VAR
	iCount		: INT;
	apply_on	: BOOL;
END_VAR
    Rectangle (127,314 451x90)
    Rectangle (578,0 127x404)
    Rectangle (127,83 451x231)
    Rectangle (127,0 451x83)
    Rectangle (0,0 127x404)
    Label (134,42 113x38), "Производитель- ность, 0-100 %"
    Label (362,42 103x34), "Скорость ТЯУ, 0-100 %"
    RoundedRectangle (472,45 80x32), "%.1f", text variable: REG_ED.Speed
        OnMouseClick: write the text variable via VisuDialogs.Numpad, min QM_MIN, max QM_MAX, title "Производительность, %"
        OnMouseClick: execute { apply_on:=TRUE; }
    RoundedRectangle (31,14 80x32), "%.1f", text variable: REG_ED.TEMPS[0]
        OnMouseClick: write the text variable via VisuDialogs.Numpad, min T_MINS_ZAD[0], max T_MAXS_ZAD[0], title "ТЕМПЕРАТУРА 1 ЗОНЫ"
        OnMouseClick: execute { apply_on:=TRUE; }
    Label (4,17 40x20), "T1"
    RoundedRectangle (31,57 80x32), "%.1f", text variable: REG_ED.TEMPS[1]
        OnMouseClick: write the text variable via VisuDialogs.Numpad, min T_MINS_ZAD[1], max T_MAXS_ZAD[1], title "ТЕМПЕРАТУРА 2 ЗОНЫ"
        OnMouseClick: execute { apply_on:=TRUE; }
    Label (4,60 40x20), "T2"
    RoundedRectangle (31,100 80x32), "%.1f", text variable: REG_ED.TEMPS[2]
        OnMouseClick: write the text variable via VisuDialogs.Numpad, min T_MINS_ZAD[2], max T_MAXS_ZAD[2], title "ТЕМПЕРАТУРА 3 ЗОНЫ"
        OnMouseClick: execute { apply_on:=TRUE; }
    Label (4,103 40x20), "T3"
    RoundedRectangle (31,143 80x32), "%.1f", text variable: REG_ED.TEMPS[3]
        OnMouseClick: write the text variable via VisuDialogs.Numpad, min T_MINS_ZAD[3], max T_MAXS_ZAD[3], title "ТЕМПЕРАТУРА 4 ЗОНЫ"
        OnMouseClick: execute { apply_on:=TRUE; }
    Label (4,146 40x20), "T4"
    RoundedRectangle (31,186 80x32), "%.1f", text variable: REG_ED.TEMPS[4]
        OnMouseClick: write the text variable via VisuDialogs.Numpad, min T_MINS_ZAD[4], max T_MAXS_ZAD[4], title "ТЕМПЕРАТУРА 5 ЗОНЫ"
        OnMouseClick: execute { apply_on:=TRUE; }
    Label (4,189 40x20), "T5"
    RoundedRectangle (31,229 80x32), "%.1f", text variable: REG_ED.TEMPS[5]
        OnMouseClick: write the text variable via VisuDialogs.Numpad, min T_MINS_ZAD[5], max T_MAXS_ZAD[5], title "ТЕМПЕРАТУРА 6 ЗОНЫ"
        OnMouseClick: execute { apply_on:=TRUE; }
    Label (4,232 40x20), "T6"
    RoundedRectangle (31,272 80x32), "%.1f", text variable: REG_ED.TEMPS[6]
        OnMouseClick: write the text variable via VisuDialogs.Numpad, min T_MINS_ZAD[6], max T_MAXS_ZAD[6], title "ТЕМПЕРАТУРА 7 ЗОНЫ"
        OnMouseClick: execute { apply_on:=TRUE; }
    Label (4,275 40x20), "T7"
    RoundedRectangle (31,315 80x32), "%.1f", text variable: REG_ED.T_MASS
        OnMouseClick: write the text variable via VisuDialogs.Numpad, min T_MIN_MASS_ZAD, max T_MAX_MASS_ZAD, title "ТЕМПЕРАТУРА РАСПЛАВА"
        OnMouseClick: execute { apply_on:=TRUE; }
    Label (4,318 40x20), "TР *"
    RoundedRectangle (31,359 80x32), "%.1f", text variable: REG_ED.T_CHIL
        OnMouseClick: write the text variable via VisuDialogs.Numpad, min T_MIN_CHIL_ZAD, max T_MAX_CHIL_ZAD, title "ТЕМПЕРАТУРА ЧИЛЛЕРА"
        OnMouseClick: execute { apply_on:=TRUE; }
    Label (4,365 40x20), "TЧ"
    RoundedRectangle (251,45 80x32), "%.1f", text variable: REG_ED.Qm
        OnMouseClick: write the text variable via VisuDialogs.Numpad, min QM_MIN, max QM_MAX, title "Производительность, %"
        OnMouseClick: execute { apply_on:=TRUE; }
    Button (594,16 96x40), "Создать новый", text variable: REG_W.Name
        OnMouseClick: execute { REG_ED:=REG_DEF; apply_on:=TRUE; }
    Button (594,82 96x40), "Загрузить", text variable: REG_W.Name, input disabled if: NOT MMCMounted
        OnMouseClick:  Dialog=DlgRegLoad, Parameters={bExtEdit: TRUE, pReg: ADR (REG_ED)}, OpenModal=True, OpenCentered=True
        OnMouseClick: execute { apply_on:=TRUE; }
        OnMouseDown: execute {
            iCount:=RECS_SELECT (0, ADR (TBL.Recs), ADR (TBL.NumFileRecs));
            IF iCount > 0 THEN
            	TBL.RowCount:=iCount;
            	TBL.RowSel:=-32768;			// Сброс выбора строки
            	TBL.PageNum:=0;				// Начальная страница
            	TBL.iMsg:=0;				// Флаг ошибок загрузки
            ELSE
            	TBL.RowCount:=0;
            	TBL.RowSel:=-32768;			// Сброс выбора строки
            	TBL.PageNum:=0;				// Начальная страница
            	CASE iCount OF
            		0: TBL.iMsg:=0; 		// Список режимов пуст
            		-1: TBL.iMsg:=1; 		// Ошибка открытия файла
            		-2: TBL.iMsg:=2; 		// Носитель не смонтирован
            	END_CASE
            END_IF
        }
    Button (594,214 96x40), "Сохранить", text variable: REG_W.Name, input disabled if: NOT MMCMounted
        OnMouseClick: execute {
            IF RECORD_SAVE (ADR (REG_ED)) THEN
            	iMsgShowDlg:=4;		// Запись успешно сохранена
            ELSE
            	iMsgShowDlg:=3;		// Ошибка сохранения
            END_IF
            CURRENT_PRG.bShowDialog:=TRUE;
        }
    Button (594,280 96x40), "Сохранить как", input disabled if: NOT MMCMounted
        OnMouseClick:  Dialog=DlgKeyboard, Parameters={ilen: , iStrLen: 63, bw: , sResult: REG_ED.Name, bShift: }, OpenModal=True, OpenCentered=True
        OnMouseDown: execute { pTargetReg:=ADR (REG_ED); }
    Button (594,350 96x40), "Применить", text variable: REG_W.Name, input disabled if: NOT apply_on
        OnMouseClick: execute {
            IF IsRegValid (ADR (REG_ED)) THEN
            	REG_W:=REG_ED;
            	AsdaSetParams ();
            	apply_on:=FALSE;
            END_IF
        }
    Label (134,98 91x24), "Частота, Гц"
    RoundedRectangle (251,92 60x32), "%.2f", text variable: REG_ED.Freq
        OnMouseClick: write the text variable via VisuDialogs.Numpad, min FREQ_MIN, max FREQ_MAX, title "ЧАСТОТА ГОЛОВКИ, Гц"
        OnMouseClick: execute { apply_on:=TRUE; }
        OnDialogClosed: execute { AsdaSetParams (); }
    Label (134,140 102x34), "ds вперёд, со знаком, мм"
    RoundedRectangle (251,142 60x32), "%.2f", text variable: REG_ED.Period.Offsets[0]
        OnMouseClick: write the text variable via VisuDialogs.Numpad, min Setts.REP_MM + 0.3, max WORK_SIZE + Setts.REP_MM - 0.3, title "ПЕРЕМЕЩЕНИЕ 1-ГО П/П"
        OnMouseClick: execute { apply_on:=TRUE; }
        OnDialogClosed: execute { AsdaSetParams (); }
    RoundedRectangle (472,142 60x32), "%.2f", text variable: REG_ED.Period.Offsets[1]
        OnMouseClick: write the text variable via VisuDialogs.Numpad, min Setts.REP_MM + 0.3, max WORK_SIZE + Setts.REP_MM - 0.3, title "ПЕРЕМЕЩЕНИЕ 2-ГО П/П"
        OnMouseClick: execute { apply_on:=TRUE; }
        OnDialogClosed: execute { AsdaSetParams (); }
    Label (363,140 102x34), "ds назад, со знаком, мм"
    Label (134,184 102x38), "Первый полупериод, %"
    RoundedRectangle (251,183 60x32), "%.2f", text variable: REG_ED.Period.Per_FirstHP
        OnMouseClick: write the text variable via VisuDialogs.Numpad, min ASDA_HP_MIN, max ASDA_HP_MAX, title "ПЕРВЫЙ ПОЛУПЕРИОД"
        OnMouseClick: execute { apply_on:=TRUE; }
        OnDialogClosed: execute { AsdaSetParams (); }
    Label (363,180 108x36), "Второй * полупериод, %"
    RoundedRectangle (472,183 60x32), "%.2f", text variable: 100 - REG_ED.Period.Per_FirstHP
    Label (134,226 75x39), "Импульс/ пауза *, %"
    RoundedRectangle (225,227 55x32), "%.2f", text variable: REG_ED.Period.Per_Pulses[0]
        OnMouseClick: write the text variable via VisuDialogs.Numpad, min ASDA_PULSE_MIN, max ASDA_PULSE_MAX, title "ИМПУЛЬС 1 ПОЛУПЕРИОДА"
        OnMouseClick: execute { apply_on:=TRUE; }
        OnDialogClosed: execute { AsdaSetParams (); }
    RoundedRectangle (450,227 55x32), "%.2f", text variable: REG_ED.Period.Per_Pulses[1]
        OnMouseClick: write the text variable via VisuDialogs.Numpad, min ASDA_PULSE_MIN, max ASDA_PULSE_MAX, title "ИМПУЛЬС 2 ПОЛУПЕРИОДА"
        OnMouseClick: execute { apply_on:=TRUE; }
        OnDialogClosed: execute { AsdaSetParams (); }
    RoundedRectangle (280,227 55x32), "%.2f", text variable: 100-REG_ED.Period.Per_Pulses[0]
    Label (364,226 75x39), "Импульс/ пауза*, %"
    RoundedRectangle (505,227 55x32), "%.2f", text variable: 100-REG_ED.Period.Per_Pulses[1]
    Label (134,277 102x25), "Уровень, %"
    RoundedRectangle (251,271 60x32), "%.2f", text variable: REG_ED.Period.Per_Levels[0]
        OnMouseClick: write the text variable via VisuDialogs.Numpad, min ASDA_LEVEL_MIN, max ASDA_LEVEL_MAX, title "УРОВЕНЬ ПЕРВОГО П/П"
        OnMouseClick: execute { apply_on:=TRUE; }
        OnDialogClosed: execute { AsdaSetParams (); }
    RoundedRectangle (472,271 60x32), "%.2f", text variable: REG_ED.Period.Per_Levels[1]
        OnMouseClick: write the text variable via VisuDialogs.Numpad, min ASDA_LEVEL_MIN, max ASDA_LEVEL_MAX, title "УРОВЕНЬ ВТОРОГО П/П"
        OnMouseClick: execute { apply_on:=TRUE; }
        OnDialogClosed: execute { AsdaSetParams (); }
    Label (364,277 97x25), "Уровень, %"
    RoundedRectangle (136,326 80x20), "Connect", colour toggle: Asda.Connect
    RoundedRectangle (400,326 80x20), "Alarm Reset", colour toggle: Asda.P4_07.1
    RoundedRectangle (488,326 80x20), "Servo ON", colour toggle: Asda.P4_07.0
    RoundedRectangle (312,326 80x20), "Reverse LIM", colour toggle: Asda.P4_07.2
    RoundedRectangle (224,326 80x20), "Forward LIM", colour toggle: Asda.P4_07.3
    Button (136,359 80x32), "Homing", input disabled if: NOT Asda.WAIT OR Asda.Block
        OnMouseClick:  Dialog=DlgConfirmAsdaCMD, Parameters={fcmd: wcAsda_Homing}, OpenModal=True, OpenCentered=True
    Button (400,359 80x32), "Парковка", input disabled if: NOT Asda.WAIT OR Asda.Block
        OnMouseClick:  Dialog=DlgConfirmAsdaCMD, Parameters={fcmd: wcAsda_Parking}, OpenModal=True, OpenCentered=True
    Button (488,359 80x32), "Работа", input disabled if: NOT Asda.WAIT OR Asda.Block
        OnMouseClick:  Dialog=DlgConfirmAsdaCMD, Parameters={fcmd: wcAsda_Working}, OpenModal=True, OpenCentered=True
    Button (224,359 80x32), "<<< Вперед", input disabled if: NOT Asda.WAIT OR Asda.Block
        OnMouseClick:  Dialog=DlgConfirmAsdaCMD, Parameters={fcmd: wcAsda_Forward}, OpenModal=True, OpenCentered=True
    Button (312,359 80x32), "Назад >>>", input disabled if: NOT Asda.WAIT OR Asda.Block
        OnMouseClick:  Dialog=DlgConfirmAsdaCMD, Parameters={fcmd: wcAsda_Backward}, OpenModal=True, OpenCentered=True
    Line (126,133) (578,133)
    Line (353,83) (352,314)
    Label (134,12 103x26), "Имя *"
    RoundedRectangle (251,6 301x32), "%s", text variable: REG_ED.Name
    Button (594,148 96x40), "Загрузить текущий", text variable: REG_W.Name, input disabled if: NOT MMCMounted
        OnMouseClick: execute { REG_ED:=REG_W; apply_on:=TRUE; }
        OnMouseDown: execute {
            iCount:=RECS_SELECT (0, ADR (TBL.Recs), ADR (TBL.NumFileRecs));
            IF iCount > 0 THEN
            	TBL.RowCount:=iCount;
            	TBL.RowSel:=-32768;			// Сброс выбора строки
            	TBL.PageNum:=0;				// Начальная страница
            	TBL.iMsg:=0;				// Флаг ошибок загрузки
            ELSE
            	TBL.RowCount:=0;
            	TBL.RowSel:=-32768;			// Сброс выбора строки
            	TBL.PageNum:=0;				// Начальная страница
            	CASE iCount OF
            		0: TBL.iMsg:=0; 		// Список режимов пуст
            		-1: TBL.iMsg:=1; 		// Ошибка открытия файла
            		-2: TBL.iMsg:=2; 		// Носитель не смонтирован
            	END_CASE
            END_IF
        }
END_VISUALIZATION

// Device/Application/Visu/DlgDeleteRec
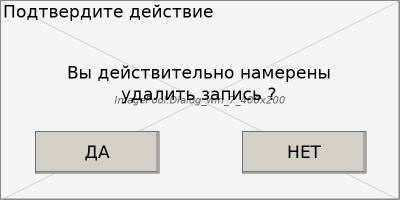
VISUALIZATION DlgDeleteRec  // 400x200
VAR_IN_OUT
END_VAR
VAR
	i_count	: INT;
END_VAR
    Image (0,0 400x200), image: ImagePool.Dialog_win_7_400x200
    Button (35,131 124x42), "ДА"
        OnMouseClick:  Dialog=DlgDeleteRec, Result=OK, NumpadKeypadSet=True
        OnMouseClick: execute {
            i_count:=REC_DELETE (ADR (TBL.Recs[TBL.RowSel]));
            TBL.RowCount:=0;
            IF i_count > 0 THEN
            	IF ((i_count-1) / TABLE_NUM_ROWS) < TBL.PageNum THEN
            		TBL.PageNum:=TBL.PageNum - 1;
            	END_IF
            	TBL.RowCount:=RECS_SELECT (TBL.PageNum * TABLE_NUM_ROWS,
            		ADR (TBL.Recs), ADR (TBL.NumFileRecs));
            	IF TBL.RowSel > (TBL.RowCount-1) THEN
            		TBL.RowSel:=TBL.RowCount-1;
            	END_IF
            ELSE
            	TBL.RowSel:=-32768;
            END_IF
        }
    Button (242,131 124x42), "НЕТ"
        OnMouseClick:  Dialog=DlgDeleteRec, Result=Cancel, NumpadKeypadSet=True
    Label (7,55 384x57), "Вы действительно намерены удалить запись ?"
    Label (0,0 248x27), "Подтвердите действие"
END_VISUALIZATION

(* text list AsdaTextList (id | default)
  0 | Ожидание команды
  1 | Инициализация сервопривода
  2 | Поиск реперной точки (Homing)
  3 | Формирование каркаса
  4 | Операция отладочного перемещения
  5 | Операция задержки
  6 | Включение сервопривода
  7 | Экстренный останов
  8 | Отключение сервопривода
  9 | Установка параметров сервопривода
  10 | Обработка ошибки
  11 | Перемещение в реперную точку
  12 | Ожидание соединения
   |  *)

(* text list AG_DVP (id | default)
  10 | Нулевая скорость движения заготовки
  9 | Превышено время движения ножа
  8 | Превышено время схода каретки с исходного концевика
  7 | РЕЗЕРВ
  6 | Каретка в крайнем положении
  5 | Превышено время возврата каретки на исходный концевик
  4 | Превышено время схода ножа с исходного концевика
  3 | Превышено время движения зажима
  2 | Нож не на исходном концевике
  1 | Зажим не на исходном концевике
  0 | Каретка не на исходном концевике
   |  *)

(* text list DvpTextList (id | default)
  0 | Система в исходном состоянии
  1 | Система в режиме РАЗОГРЕВ
  2 | Система в рабочем состоянии
  3 | Система в режиме выгона массы
   |  *)

(* text list AG_CONNECT (id | default)
  4 | Нет соединения с Чиллером
  3 | Нет соединения с ПЧВ тянущего устройства
  2 | Нет соединения с ПЧВ шнека
  1 | Нет соединения с контроллером DVP
  0 | Нет соединение с сервоприводом ASDA-A2
   |  *)

(* text list MSGS (id | default)
  13 | Низкий уровень воды в баке !!!
  12 | Перегрев ПЧВ тянущего устройства
  11 | Перегрузка по току ПЧВ тянущего устройства
  10 | Напряжение не в норме ПЧВ тянущего устройства
  9 | Предупреждение от ПЧВ тянущего устройства
  8 | Перегрев ПЧВ шнека
  7 | Перегрузка по току ПЧВ шнека
  6 | Напряжение не в норме ПЧВ шнека
  5 | Предупреждение от ПЧВ шнека
  4 | Низкое давление воздуха !!!
  3 | Низкий уровень сырья в бункере !!!
  2 | Выведите бункер !!!
  1 | Бункер выведен !!!
  0 | Система вышла на режим !
   |  *)

(* text list AG_AVAR (id | default)
  4 | 
  3 | Низкая температура одной из зон
  2 | Превышена температура одной из зон
  1 | Температура одной из зон ниже температуры запуска привода
  0 | Превышена критическая температура одной из зон
   |  *)

(* text list AG_DEV (id | default)
  11 | Тестовая авария
  13 | Авария Чиллера
  10 | Аварийный сигнал ПЧВ тянущего устройства
  7 | Аварийный сигнал ПЧВ шнека
  6 | Тестовая ошибка
  5 | Превышено время операции отладки
  4 | РЕЗЕРВ АВАРИИ
  3 | Превышено время операции HOMING
  2 | Ошибка инициализации Р2-30 или Р3-06
  1 | Сигнал предупреждения от сервопривода
  0 | Сигнал аварии от сервопривода
   |  *)

(* text list AG_CHILLER (id | default)
  35 | Авария Чиллера
  34 | Неисправен датчик элетрического сопротивления жидкости в Чиллере
  33 | Повышение элетрического удельного сопротивления жидкости в Чиллере
  32 | Обнаружена утечка воды Чиллера
  31 | Обнаружен сигнал контакта входа 2 Чиллера
  30 | Обнаружен сигнал контакта входа 1 Чиллера
  29 | Обслуживание компрессора двигателя Чиллера
  28 | Обслуживание вентилятора двигателя Чиллера
  27 | Обслуживание насоса Чиллера
  26 | Неисправность датчика давления на входе компрессора Чиллера
  25 | Неисправность датчика давления нагнетания компрессора Чиллера
  24 | Неисправность датчика давления нагнетания Чиллера
  23 | Неисправность датчика температуры на входе компрессора Чиллера
  22 | Неисправность датчика температуры на входе Чиллера
  21 | Неисправность датчика температуры на выходе Чиллера
  20 | Сработал предохранитель постоянного тока в Чиллере
  19 | Ошибка памяти контроллера Чиллера
  18 | Ошибка связи с контроллером Чиллера
  17 | Перегрузка компрессора Чиллера
  16 | Падение давления на низкой стороне контура хладагента Чиллера
  15 | Повышение давления на низкой стороне контура хладагента Чиллера
  14 | Падение давления на высокой стороне контура хладагента Чиллера
  13 | Unused
  12 | Высокое давление нагнетания компрессора Чиллера
  11 | Низкая температура нагревания Чиллера
  10 | Низкая температура на входе компрессора Чиллера
  9 | Высокая температура на входе компрессора Чиллера
  8 | Падение давления нагнетания Чиллера
  7 | Повышение давления нагнетания Чиллера
  6 | Ненормальная работа насоса Чиллера
  5 | Высокая давление нагнетания Чиллера
  4 | Высокая температура воды на входе Чиллера
  3 | Температура на выходе Чиллера...
  2 | Температура на выходе Чиллера выросла
  1 | Высокая температура воды на выходе Чиллера
  0 | Низкий уровень воды в Чиллере
   |  *)

(* text list FileTextList (id | default)
  0 | Список режимов пуст !!!
  1 | Не смонтирован флеш-носитель !!!
  2 | Ошибка открытия файла !!!
  3 | Ошибка сохранения !!!
  4 | Запись успешно сохранена
  5 | Настройки успешно сохранены
  6 | Ошибка при сохранении настроек
  7 | Настройки успешно загружены
  8 | Ошибка при загрузке настроек
   |  *)
